FUNCTION_BLOCK CvToGTranslator
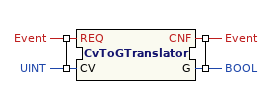
  EVENT_INPUT
    REQ WITH CV;
  END_EVENT
  EVENT_OUTPUT
    CNF WITH G;
  END_EVENT
  VAR_INPUT
    CV : UINT;
  END_VAR
  VAR_OUTPUT
    G : BOOL;
  END_VAR
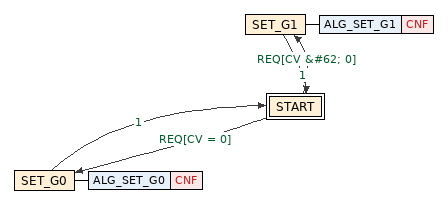
  EC_STATES
    START;
    SET_G1 : ALG_SET_G1 -> CNF;
    SET_G0 : ALG_SET_G0 -> CNF;
  END_STATES
  EC_TRANSITIONS
    START TO SET_G1 := REQ[CV &#62; 0];
    START TO SET_G0 := REQ[CV = 0];
    SET_G1 TO START := 1;
    SET_G0 TO START := 1;
  END_TRANSITIONS
  ALGORITHM ALG_SET_G1 IN ST:

  END_ALGORITHM
  ALGORITHM ALG_SET_G0 IN ST:

  END_ALGORITHM
END_FUNCTION_BLOCK
